TEXTLIST TL_TctrlPowerTerminal
  0 = 'NoTerminal'
  1 = 'KL3403'
  2 = 'EL3403'
  3 = 'EL3773'
  4 = 'EL3x64'
  1000 = 'Simualtion'
  10000 = 'Customized'
   = ''
END_TEXTLIST

(* stored: Version 1.1.0.1, ProductVersion 3.1.4018.5
   TextList TL_TctrlPowerTerminal: Id {24ab8e47-3432-4625-b110-b881a322190c} *)
